// TIA Portal V20 export
TYPE "LER_typeReadWriteUDT"
// stored: Access Published
   STRUCT
      Input : Struct
         execute : Bool;
         addrTag : DWord;
         lengthData : Word;
      END_STRUCT;
      Output : Struct
         done : Bool;
         busy : Bool;
         error : Bool;
         status : DWord;
         pressence : Bool;
      END_STRUCT;
      InOut : Struct
         rfidData : Array[0..255] of Byte;
      END_STRUCT;
   END_STRUCT;
END_TYPE
